FUNCTION_BLOCK linear_trajectory_with_quintic_polynomial_blends
VAR_INPUT
	t0,t1,q0,q1:lreal;
	t:lreal;	
END_VAR
VAR_OUTPUT
	pos:lreal;
	vel:lreal;
	acc:lreal;
	finished:BOOL;
END_VAR
VAR
	h,Tp,ratio,TS,TA:lreal;
	k1,t_qa,t_qb,qa,qb:lreal;
	
	Quintic_spline_curve_factor_1:Quintic_spline_curve_factor;
	Quintic_spline_curve_factor_2:Quintic_spline_curve_factor;
	a0,a1,a2,a3,a4,a5:ARRAY[1..2] OF lreal;	
END_VAR


h:=q1-q0;
Tp:=t1-t0;

ratio:=0.15;
Ts:=Tp*ratio;
Ta:=2*Ts;

k1:=h/(t1-t0-2*Ts);
t_qa:=t0+Ta;  qa:=q0+k1*(t_qa-(t0+Ts));
t_qb:=t1-Ta;  qb:=q0+k1*(t_qb-(t0+Ts));


//%计算第1段轨迹,五次多项式，始末位置的速度、加速度都为零
Quintic_spline_curve_factor_1(
	t0:= t0, 
	t1:= t_qa, 
	q0:= q0, 
	q1:= qa, 
	v0:= 0, 
	v1:= k1, 
	acc0:= 0, 
	acc1:= 0, 
	a0=> a0[1], 
	a1=> a1[1], 
	a2=> a2[1], 
	a3=> a3[1], 
	a4=> a4[1], 
	a5=> a5[1]);


//%计算第2段轨迹，直线




//%计算第3段轨迹，五次多项式，始末位置的速度、加速度都为零
Quintic_spline_curve_factor_2(
	t0:= t_qb, 
	t1:= t1, 	
	q0:= qb, 
	q1:= q1, 
	v0:= k1, 
	v1:= 0, 
	acc0:= 0, 
	acc1:= 0, 
	a0=> a0[2], 
	a1=> a1[2], 
	a2=> a2[2], 
	a3=> a3[2], 
	a4=> a4[2], 
	a5=> a5[2]);


	
	
	
IF (t<=t_qa)THEN
	t0:=t0;
	pos:=a0[1]+a1[1]*(t-t0)+a2[1]*EXPT((t-t0),2)+a3[1]*EXPT((t-t0),3)+a4[1]*EXPT((t-t0),4)+a5[1]*EXPT((t-t0),5);
	vel:=a1[1]+2*a2[1]*(t-t0)+3*a3[1]*EXPT((t-t0),2)+4*a4[1]*EXPT((t-t0),3)+5*a5[1]*EXPT((t-t0),4);
    acc:=2*a2[1]+6*a3[1]*(t-t0)+12*a4[1]*EXPT((t-t0),2)+20*a5[1]*EXPT((t-t0),3);
	
ELSIF (t<=t_qb) THEN
	t0:=t_qa;
	pos:=qa+k1*(t-t0);
	vel:=k1;
	acc:=0;
	
ELSIF (t<=t1)THEN	
	t0:=t_qb;
	pos:=a0[2]+a1[2]*(t-t0)+a2[2]*EXPT((t-t0),2)+a3[2]*EXPT((t-t0),3)+a4[2]*EXPT((t-t0),4)+a5[2]*EXPT((t-t0),5);
	vel:=a1[2]+2*a2[2]*(t-t0)+3*a3[2]*EXPT((t-t0),2)+4*a4[2]*EXPT((t-t0),3)+5*a5[2]*EXPT((t-t0),4);
	acc:=2*a2[2]+6*a3[2]*(t-t0)+12*a4[2]*EXPT((t-t0),2)+20*a5[2]*EXPT((t-t0),3);
END_IF


IF (t>t1) THEN
	finished:=TRUE;
	pos:=q1;
	vel:=0;
	acc:=0;
ELSE
	finished:=FALSE;
END_IF

END_FUNCTION_BLOCK

(* stored: Version 1.1.0.1, ProductVersion 3.1.4024.12
   POU linear_trajectory_with_quintic_polynomial_blends: Id {6755b785-4d15-4568-ad5f-31f530015fcc}, SpecialFunc None *)
